TYPE Module_Palletizer_AX_OUT :
STRUCT
	;
END_STRUCT
END_TYPE

(* stored: Version 1.1.0.1, ProductVersion 3.1.4024.11
   DUT Module_Palletizer_AX_OUT: Id {86c8f9e8-6238-4882-addd-272786907fc3} *)
